FUNCTION_BLOCK ConcatStringRpcHandler IMPLEMENTS I_RpcHandler
VAR
END_VAR

METHOD Handle
VAR_INPUT
	Parameters : I_RpcParameters;
	Reply : I_RpcSynchronousReply;
END_VAR
VAR
	str1 : T_MAXSTRING;
	str2 : T_MAXSTRING;
	result : T_MAXSTRING;
END_VAR
IF NOT Parameters.TryGetParameter('STR1',str1) THEN
	Reply.RejectWithMessage('Missing STR1 parameter');
	RETURN;
END_IF

IF NOT Parameters.TryGetParameter('STR2',str2) THEN
	Reply.RejectWithMessage('Missing STR2 parameter');
	RETURN;
END_IF

result := CONCAT(str1, str2);

Reply.Compose().AddString(result).Send();

//Reply.WithString(result).Send();
END_METHOD

END_FUNCTION_BLOCK

(* stored: Version 1.1.0.1, ProductVersion 3.1.4024.12
   POU ConcatStringRpcHandler: Id {3308dee3-7162-4e6b-ab6c-6da43be8ef3f}, SpecialFunc None
   Method Handle: Id {b973a79f-d251-4a0d-baf6-50941936d5fe} *)
